// TwinCAT 3 PLC project BaseElements
// Title: Base_Hts
// Company: Vistaprint
// Author: AVME/DSC
// ProjectVersion: 0.0.0.50
// Description: 0.0.0.50 - HFE: Bug fixed 0.0.0.49 - HFE: desable of last station 0.0.0.48 - Add AutoMode to HRU 0.0.0.47 - Some Bugs in DPJ fixed 0.0.0.46 - BaseElements 0.0.1.18 Some Bugs in DPJ, JUN fixed 0.0.0.45 - BaseElements 0.0.1.17 MTR/sta_RUN Bug fixed 0.0.0.44 - New Libs BasePLC 0.3.4.8, BaseElements 0.0.1.16 0.0.0.43 - DPJ reworked (Missed Shirt Problem) 0.0.0.42 - MER - new parameter added HFE reworked 0.0.0.41 - BasePLC V0.3.4.5; BaseElements V0.0.1.9 0.0.0.40 - Add MTR Parameter dinWaitBetweenSensorAndReservation_um 0.0.0.39 - Bug fixed in HFE, CHD; FOC and FOD added 0.0.0.34 - JUN / DPJ replaced with version from Shirtstream 0.0.0.32 - HFE from Lvl1 to Lvl2 and reworked 0.0.0.30 - BaseElements 0.0.1.5 BasePLC 0.3.4.3 included, Tc2_SerialCom 0.0.0.29 - BaseElements 0.0.1.2 BasePLC 0.3.4.2 included; FB_CtrlModule moved to BaseElements 0.0.0.28 - Added ADS data channel to FB_HPS for shirt request from Heatpress 0.0.0.27 - Added bolStopReleaseHangers 0.0.0.26 - DPJ.sta_RUN Entry action reworked 0.0.0.25 - Error JUN changed 0.0.0.24 - Rising Edge detection of bolBringShirt in HPS 0.0.0.23 - HTS, hanger turned line wait at SEP 0.0.0.22 - Bug fixed in STOPbusy 0.0.0.21 - Bugs fixed in HPS 0.0.0.20 - HPS with new Child SEP New BaseElements 0.0.0.20 0.0.0.19 - Alternativ status for run sequence added; Timing reworked in MER jam detection; DPJ STOPBusy reworked, HRU Errors reworked, DPJ new Errors 12 and 13 added 0.0.0.18 - Timeout Run / Stop sequence added 0.0.0.17 - EMO reworked in BaseCtrlModule; CHD "destination full" reworked; AddStpGrp, AddRunGrp removed 0.0.0.16 - Back to BasePLC Lib. V3.3.5 beacuase of PageFaults 0.0.0.15 - Rebuild 0.0.0.14 - Bugzilla ID 03: BufferFull for LineControl added 0.0.0.13 - Bugzilla ID 55: reworked refill of SLB/STB 0.0.0.12 - Update of BasePLC 0.3.3.7, BaseElements 0.0.0.17 0.0.0.11 - Add more controllers to the library (LAI, CHD, HFE, PLS, JUN, DPJ, MER, HRU, HPS, COS, STB, SLB) 0.0.0.10 - Clear pending command to prevent automatic recovery in sta_STOPBusy 0.0.0.9 - BugFix in sub state "cSTA_SUB_CHECK_GROUP_STATUS" from run and stop sequence. Insert new "bolChecked" flag to detect if the sequence has been processed correctly. 0.0.0.8 - Add TSTOP in checkChildAlmClass 0.0.0.7- General revision of behaviour in case of emergency off (state EOFF) and general error (state ERROR). New handling for module specific interface. 0.0.0.6 - Go to EOFFBusy if not in sta_EOFF 0.0.0.5 - In Always: go to EOFFBusy at generalFault 0.0.0.4 - In Always: go to EOFFBusy not to EOFF at emergency stop 0.0.0.3 - Remove CurrentItemCounter and his inputs 0.0.0.2 - Changes after first use in simulation in ICL Module 0.0.0.1 - First release
// ProgramVersion: 3.1.0.5
// libraries:
//   Base_Elements,0.0.1.18,Vistaprint
//   Base_PLC,0.3.4.8,Vistaprint
//   Tc2_Standard,3.3.0.0,Beckhoff Automation GmbH
//   Tc2_System,3.3.5.0,Beckhoff Automation GmbH
//   Tc2_Utilities,3.3.7.0,Beckhoff Automation GmbH
//   Tc3_Module,3.3.5.0,Beckhoff Automation GmbH
// project tree:
//   POUs/Controller/Driver/FOD/ FB_ReceiveFolderState.TcPOU (not stored), FB_SendFolderMessage.TcPOU, T_FOD.TcDUT (not stored), T_FOD_Cfg.TcDUT (not stored), T_FOD_Cur.TcDUT (not stored), T_FOD_StateMachine.TcDUT (not stored)
//   POUs/Controller/Driver/FOD/Infrastructure/ FB_DecodeCanRxMessage.TcPOU (not stored), fb_GenerateCanTxMessage.TcPOU
//   POUs/Controller/Lvl0/CHD %28Cross Hanger Detection%29/ CHD_CmdState.TcGVL (not stored), Const_CHD.TcGVL (not stored), FB_CHD.TcPOU (not stored), T_CheckElement.TcDUT (not stored), T_Ctrl_SIf_CHD.TcDUT (not stored), T_Ctrl_SIf_CHD_Cfg.TcDUT (not stored), T_Ctrl_SIf_CHD_Cur.TcDUT (not stored), T_Ctrl_SIf_CHD_In.TcDUT (not stored), T_Ctrl_SIf_CHD_Out.TcDUT (not stored), T_Ctrl_SIf_CHD_Par.TcDUT (not stored)
//   POUs/Controller/Lvl0/FOC %28Folder Communication%29/ FB_FOC.TcPOU (not stored), FOC_CmdState.TcGVL (not stored), T_Ctrl_SIf_FOC.TcDUT (not stored), T_Ctrl_SIf_FOC_Cfg.TcDUT (not stored), T_Ctrl_SIf_FOC_Cur.TcDUT (not stored), T_Ctrl_SIf_FOC_In.TcDUT (not stored), T_Ctrl_SIf_FOC_Out.TcDUT (not stored), T_Ctrl_SIf_FOC_Par.TcDUT (not stored)
//   POUs/Controller/Lvl0/HRU %28Hanger Rotation Unit%29/ FB_HRU.TcPOU (not stored), HRU_CmdState.TcGVL (not stored), T_Ctrl_SIf_HRU.TcDUT (not stored), T_Ctrl_SIf_HRU_In.TcDUT (not stored), T_Ctrl_SIf_HRU_Out.TcDUT (not stored), T_Ctrl_SIf_HRU_Par.TcDUT (not stored)
//   POUs/Controller/Lvl0/JUN %28Junction%29/ E_Typ_JUN.TcDUT (not stored), FB_JUN.TcPOU (not stored), JUN_CmdState.TcGVL (not stored), T_Ctrl_SIf_JUN.TcDUT (not stored), T_Ctrl_SIf_JUN_Cfg.TcDUT (not stored), T_Ctrl_SIf_JUN_Cur.TcDUT (not stored), T_Ctrl_SIf_JUN_Ilk.TcDUT (not stored), T_Ctrl_SIf_JUN_In.TcDUT (not stored), T_Ctrl_SIf_JUN_Out.TcDUT (not stored), T_Ctrl_SIf_JUN_Par.TcDUT (not stored), T_JUN_OutfeedCheck.TcDUT (not stored)
//   POUs/Controller/Lvl0/LAI %28Labler Interface%29/ FB_LAI.TcPOU (not stored), T_Ctrl_SIf_LAI.TcDUT (not stored), T_Ctrl_SIf_LAI_Cfg.TcDUT (not stored), T_Ctrl_SIf_LAI_Cur.TcDUT (not stored), T_Ctrl_SIf_LAI_In.TcDUT (not stored), T_Ctrl_SIf_LAI_Out.TcDUT (not stored), T_Ctrl_SIf_LAI_Par.TcDUT (not stored)
//   POUs/Controller/Lvl0/PLS %28PickToLight System%29/ Const_PLS.TcGVL (not stored), FB_PLS.TcPOU (not stored), T_Ctrl_SIf_PLS.TcDUT (not stored), T_Ctrl_SIf_PLS_Cfg.TcDUT (not stored), T_Ctrl_SIf_PLS_Cur.TcDUT (not stored), T_Ctrl_SIf_PLS_In.TcDUT (not stored), T_Ctrl_SIf_PLS_Out.TcDUT (not stored), T_Ctrl_SIf_PLS_Par.TcDUT (not stored)
//   POUs/Controller/Lvl0/STB %28Stopper buffer%29/ FB_STB.TcPOU (not stored), STB_CmdState.TcGVL (not stored), T_Ctrl_SIf_STB.TcDUT (not stored), T_Ctrl_SIf_STB_Cfg.TcDUT (not stored), T_Ctrl_SIf_STB_Cur.TcDUT (not stored), T_Ctrl_SIf_STB_Ilk.TcDUT (not stored), T_Ctrl_SIf_STB_In.TcDUT (not stored), T_Ctrl_SIf_STB_Out.TcDUT (not stored), T_Ctrl_SIf_STB_Par.TcDUT (not stored)
//   POUs/Controller/Lvl1/DPJ %28DecisionPoint Junction%29/ Const_DPJ.TcGVL (not stored), DPJ_CmdState.TcGVL (not stored), E_DecisionState.TcDUT (not stored), E_Decision_Job.TcDUT (not stored), E_ProductFlowState.TcDUT (not stored), FB_DPJ.TcPOU (not stored), FB_DtChnToLine_JobDone.TcPOU (not stored), T_Ctrl_SIf_DPJ.TcDUT (not stored), T_Ctrl_SIf_DPJ_Cfg.TcDUT (not stored), T_Ctrl_SIf_DPJ_Cur.TcDUT (not stored), T_Ctrl_SIf_DPJ_DtChnToLine.TcDUT (not stored), T_Ctrl_SIf_DPJ_DtChnToPLC.TcDUT (not stored), T_Ctrl_SIf_DPJ_In.TcDUT (not stored), T_Ctrl_SIf_DPJ_Out.TcDUT (not stored), T_Ctrl_SIf_DPJ_Par.TcDUT (not stored), T_Decision.TcDUT (not stored), T_DecisionElement.TcDUT (not stored), T_Decision_DtChn.TcDUT (not stored), T_JobDone_DtChn.TcDUT (not stored), T_SimDtChn.TcDUT (not stored)
//   POUs/Controller/Lvl1/SLB %28Slide buffer%29/ Const_SLB.TcGVL (not stored), FB_SLB.TcPOU (not stored), SLB_CmdState.TcGVL (not stored), T_Ctrl_SIf_SLB.TcDUT (not stored), T_Ctrl_SIf_SLB_Cfg.TcDUT (not stored), T_Ctrl_SIf_SLB_Cur.TcDUT (not stored), T_Ctrl_SIf_SLB_In.TcDUT (not stored), T_Ctrl_SIf_SLB_Par.TcDUT (not stored)
//   POUs/Controller/Lvl2/COS %28Control Station%29/ COS_CmdState.TcGVL (not stored), FB_COS.TcPOU (not stored), T_Ctrl_SIf_COS.TcDUT (not stored), T_Ctrl_SIf_COS_Cfg.TcDUT (not stored), T_Ctrl_SIf_COS_Cur.TcDUT (not stored), T_Ctrl_SIf_COS_In.TcDUT (not stored), T_Ctrl_SIf_COS_Par.TcDUT (not stored)
//   POUs/Controller/Lvl2/FOL %28Folder%29/ FB_FOL.TcPOU (not stored), FOL_CmdState.TcGVL (not stored), T_Ctrl_SIf_FOL.TcDUT (not stored), T_Ctrl_SIf_FOL_Cfg.TcDUT (not stored), T_Ctrl_SIf_FOL_Cur.TcDUT (not stored), T_Ctrl_SIf_FOL_In.TcDUT (not stored), T_Ctrl_SIf_FOL_Out.TcDUT (not stored), T_Ctrl_SIf_FOL_Par.TcDUT (not stored)
//   POUs/Controller/Lvl2/HFE/ Const_HFE.TcGVL, FB_HFE.TcPOU, T_Ctrl_SIf_HFE.TcDUT, T_Ctrl_SIf_HFE_Cfg.TcDUT, T_Ctrl_SIf_HFE_Cur.TcDUT, T_Ctrl_SIf_HFE_Par.TcDUT
//   POUs/Controller/Lvl2/HPS %28Heat Press Shirt Station%29/ Const_HPS.TcGVL (not stored), E_DtChnJob.TcDUT (not stored), FB_DtChnToLine_ChargeDone.TcPOU (not stored), FB_HPS.TcPOU (not stored), T_ChargeDone_DtChn.TcDUT (not stored), T_Ctrl_SIf_HPS.TcDUT (not stored), T_Ctrl_SIf_HPS_Ads.TcDUT (not stored), T_Ctrl_SIf_HPS_Ads_Read.TcDUT (not stored), T_Ctrl_SIf_HPS_Cfg.TcDUT (not stored), T_Ctrl_SIf_HPS_Cur.TcDUT (not stored), T_Ctrl_SIf_HPS_DtChnToLine.TcDUT (not stored), T_Ctrl_SIf_HPS_DtChnToPLC.TcDUT (not stored), T_Ctrl_SIf_HPS_In.TcDUT (not stored), T_Ctrl_SIf_HPS_Out.TcDUT (not stored), T_Ctrl_SIf_HPS_Par.TcDUT (not stored), T_NewCharge_DtChn.TcDUT (not stored)
//   POUs/Controller/Lvl2/MER %28Merger Standard%29/ Const_MER.TcGVL (not stored), E_Typ_MER_AUTO_MODE.TcDUT (not stored), E_Typ_MER_MODE.TcDUT (not stored), FB_MER.TcPOU (not stored), T_Ctrl_SIf_MER.TcDUT (not stored), T_Ctrl_SIf_MER_Cfg.TcDUT (not stored), T_Ctrl_SIf_MER_Cur.TcDUT (not stored), T_Ctrl_SIf_MER_In.TcDUT (not stored), T_Ctrl_SIf_MER_Par.TcDUT (not stored), T_Line.TcDUT (not stored)
//   POUs/Controller/Lvl2/MTR %28Merger Transport%29/ Const_MTR.TcGVL (not stored), E_Typ_MTR_SECTION_STATE.TcDUT (not stored), FB_MTR.TcPOU (not stored), T_Ctrl_SIf_MTR.TcDUT (not stored), T_Ctrl_SIf_MTR_Cfg.TcDUT (not stored), T_Ctrl_SIf_MTR_Cur.TcDUT (not stored), T_Ctrl_SIf_MTR_In.TcDUT (not stored), T_Ctrl_SIf_MTR_Par.TcDUT (not stored), T_MTR_Buffer_Sections.TcDUT (not stored)
//   Version/ Global_Version.TcGVL
// (motion and I/O tree: see PLC project basehtssample)
// real-time tasks:
//   TASK Task_Fast: cycle T#2ms, priority 3, ADS port 350
//   TASK Task_Slow: cycle T#50000us, priority 20, ADS port 351
//   TASK Task_Middle: cycle T#10ms, priority 10, ADS port 352

// ---- POUs/Controller/Lvl2/HFE/T_Ctrl_SIf_HFE.TcDUT
TYPE T_Ctrl_SIf_HFE :
STRUCT
	///configuration
	Cfg: T_Ctrl_SIf_HFE_Cfg;
	///parameter
	Par: T_Ctrl_SIf_HFE_Par;
	///current values
	Cur: T_Ctrl_SIf_HFE_Cur;
	///alarm number used in this controller
	Alm: ARRAY[1..2] OF T_Ctrl_Alm;
END_STRUCT
END_TYPE

// ---- POUs/Controller/Lvl2/HFE/T_Ctrl_SIf_HFE_Cfg.TcDUT
TYPE T_Ctrl_SIf_HFE_Cfg :
STRUCT
	/// Number of supportetd LDS
	uintNbOfLDS: UINT;
END_STRUCT
END_TYPE

// ---- POUs/Controller/Lvl2/HFE/T_Ctrl_SIf_HFE_Cur.TcDUT
TYPE T_Ctrl_SIf_HFE_Cur :
STRUCT
END_STRUCT
END_TYPE

// ---- POUs/Controller/Lvl2/HFE/T_Ctrl_SIf_HFE_Par.TcDUT
TYPE T_Ctrl_SIf_HFE_Par :
STRUCT
	// Waiting between SLB-STB Close and Junction open
	udiWaitingTime_ms: UDINT;
	// Open junction time
	a_udiTimeOpen_ms: ARRAY[0..cuintMaxStation] OF UDINT;
	// Close junction time
	a_udiTimeClose_ms: ARRAY[0..cuintMaxStation] OF UDINT;
	// Enable Junction to LDS
	a_bolEnableJunction: ARRAY[0..cuintMaxStation] OF BOOL;
END_STRUCT
END_TYPE

// ---- POUs/Controller/Lvl2/HFE/Const_HFE.TcGVL
VAR_GLOBAL CONSTANT
	cuintMaxStation: INT := 4;
END_VAR

// ---- Version/Global_Version.TcGVL
// This function has been automatically generated from the project information.
VAR_GLOBAL CONSTANT
	{attribute 'const_non_replaced'}
	stLibVersion_Base_Hts : ST_LibVersion := (iMajor := 0, iMinor := 0, iBuild := 0, iRevision := 50, sVersion := '0.0.0.50');
END_VAR

// ---- POUs/Controller/Driver/FOD/FB_SendFolderMessage.TcPOU
FUNCTION_BLOCK FB_SendFolderMessage
VAR_INPUT
	InTxCounter AT %I*: UINT;
	CpuOnline: BOOL;
	EmptyHangerConveying: BOOL;
	ProgramNumber: BYTE := 1;
	/// 1=forward, 2=sideward
	ShirtStackConveyor: BYTE := 1;
	ChangeCustomer: BOOL;
	StopFolder: BOOL;
	ShotOutStacks: BOOL;
	/// CAN Identifier of receiver
	TxCobId: UINT := 113;
	/// true = starts sending a message. make sure all data fields are set before.
	bStartSend: BOOL;
	/// timeout after sent message before next message will be send
	tTimeout: TIME := TIME#50ms;
END_VAR
VAR_OUTPUT
	TxMessages AT %Q*: ARRAY[0..9] OF CANQUEUE;
	OutTxCounter AT %Q*: UINT;
	OutNoOfTxMessages AT %Q*: UINT := 1;
END_VAR
VAR
	uinState: UINT;
	BytesToSend: UINT := 8;
	arrDataToSend: CANMESSAGE;
	m: UINT;
	fbGenerateTxMessage: fb_GenerateCanTxMessage;
	uliCountSentMessages: ULINT;
	tWaitTimer: TON;
END_VAR
VAR CONSTANT
	cSTA_WAIT_SEND: UINT := 10;
	cSTA_SEND_MESSAGE: UINT := 20;
	cSTA_WAIT_SEND_COMPLETE: UINT := 30;
	cSTA_WAIT_BEFORE_SEND_NEXT: UINT := 40;
END_VAR

(*__________________________________________________________________________________________________
¦	
¦	Vistaprint Schweiz GmbH
¦	CH - 8401 Winterthur
¦
¦	www.vistaprint.ch - info@vistaprint.ch
¦___________________________________________________________________________________________________

Function desription:
CAN communication to Kannegiesser folder to send commands.


History:
Version		Date			Author		Comment
---------------------------------------------------------------------------------------------------
0.00.1		28.09.2013		VP/RE		Start history
0.00.2		29.10.2013		VP/RE		Introduced state names
0.00.3		11.12.2013		VP/RE		Implemented sleep timeout after sending a CAN message.
___________________________________________________________________________________________________*)


CASE uinState OF
	
cSTA_WAIT_SEND:	
	IF bStartSend THEN
		bStartSend:=FALSE;
		uinState := cSTA_SEND_MESSAGE;
	END_IF
	
cSTA_SEND_MESSAGE:	
	
	uliCountSentMessages := uliCountSentMessages + 1;

	FOR m := 0 TO OutNoOfTxMessages - 1 DO
		
		arrDataToSend[0].0 := CpuOnline;
		arrDataToSend[0].1 := EmptyHangerConveying;
		arrDataToSend[1].0 := ChangeCustomer;
		
		arrDataToSend[0].4 := ProgramNumber.0;
		arrDataToSend[0].5 := ProgramNumber.1;
		arrDataToSend[0].6 := ProgramNumber.2;
		arrDataToSend[0].7 := ProgramNumber.3;
		
		IF (ShirtStackConveyor = 1) THEN
			arrDataToSend[2].1 := 1;
			arrDataToSend[2].2 := 0;
		ELSIF (ShirtStackConveyor = 2) THEN
			arrDataToSend[2].1 := 0;
			arrDataToSend[2].2 := 1;
		ELSIF (ShirtStackConveyor = 0) THEN
			arrDataToSend[2].1 := 0;
			arrDataToSend[2].2 := 0;
		END_IF
		
		arrDataToSend[3].5 := StopFolder;
		arrDataToSend[3].6 := ShotOutStacks;

		fbGenerateTxMessage(CobId := TxCobId,
							BytesToSend := BytesToSend,
							arrDataToSend := arrDataToSend ,
							TxMessage => TxMessages[0] );
	END_FOR
	
	OutTxCounter := OutTxCounter + 1;
	uinState := cSTA_WAIT_SEND_COMPLETE;
	
cSTA_WAIT_SEND_COMPLETE:	
	IF OutTxCounter = InTxCounter THEN
		uinState := cSTA_WAIT_BEFORE_SEND_NEXT;
	END_IF

cSTA_WAIT_BEFORE_SEND_NEXT:
	IF (tWaitTimer.Q = TRUE) THEN
		uinState := cSTA_WAIT_SEND;
	END_IF
	
END_CASE

tWaitTimer(IN := uinState = cSTA_WAIT_BEFORE_SEND_NEXT, PT := tTimeout);

METHOD init
uinState := cSTA_WAIT_SEND;
END_METHOD

END_FUNCTION_BLOCK

// ---- POUs/Controller/Driver/FOD/Infrastructure/fb_GenerateCanTxMessage.TcPOU
FUNCTION_BLOCK fb_GenerateCanTxMessage
VAR_INPUT
	CobId: UINT;
	BytesToSend: UINT;
	arrDataToSend: CANMESSAGE;
END_VAR
VAR_OUTPUT
	TxMessage: CANQUEUE;
END_VAR

TxMessage.CobId := (SHL(CobId,5)) + BytesToSend;
TxMessage.data := arrDataToSend;

END_FUNCTION_BLOCK

// ---- POUs/Controller/Lvl2/HFE/FB_HFE.TcPOU
FUNCTION_BLOCK FB_HFE EXTENDS FB_CtrlBase
VAR_INPUT
	a_bolLDSNeedsHanger: ARRAY[0..cuintMaxStation] OF BOOL;
	a_intHFE_BufferZone: ARRAY[0..cuintMaxStation] OF INT;
	p_fbTlpDrive: POINTER TO FB_DRV;
	///p_fbJunction : POINTER TO FB_JUN;
	p_fbSLB: POINTER TO FB_SLB;
END_VAR
VAR
	/// List of pointers to Childs of VLV
	a_pMultiChildCtrl: ARRAY[0..Base_Const.cMaxNrOfChilds] OF POINTER TO FB_VLV;
	/// List of childs common interface
	a_pMultiChildCIF: ARRAY[0..Base_Const.cMaxNrOfChilds] OF POINTER TO T_Ctrl_CIf;
	/// List of childs specific interface for additional parameters or cur
	a_pMultiChildSIF: ARRAY[0..Base_Const.cMaxNrOfChilds] OF POINTER TO Base_Elements.T_Ctrl_SIf_VLV;
	usiNumOfMultiChild: USINT;
	usiNumOfValidPointerMultiChild: USINT;
	/// Specific interface struct for public access
	SIf: T_Ctrl_SIf_HFE;
	/// Child controller
	pTlpDrive_CIf: POINTER TO T_Ctrl_CIf;
	///pJunction_CIf : POINTER TO T_Ctrl_CIf;
	pSLB_CIf: POINTER TO T_Ctrl_CIf;
	pSLB_SIf: POINTER TO T_Ctrl_SIf_SLB;
	intSubState: ARRAY[0..cuintMaxStation] OF INT;
	udiTimeInStateRefill_ms: ARRAY[0..cuintMaxStation] OF UDINT;
END_VAR
VAR CONSTANT
	/// sub States
	cSTA_SUB_WaitForJob: INT := 500;
	cSTA_SUB_WaitOpen: INT := 502;
	cSTA_SUB_Open: INT := 504;
	cSTA_SUB_WaitClose: INT := 506;
	cSTA_SUB_Close: INT := 508;
END_VAR

(*__________________________________________________________________________________________________
¦	
¦	Vistaprint Schweiz GmbH
¦	CH - 8401 Winterthur
¦
¦	www.vistaprint.ch - info@vistaprint.ch
¦___________________________________________________________________________________________________

Function desription:
Cylinder implementation. 


History:
Version		Date			Author		Comment
---------------------------------------------------------------------------------------------------
0.00.1		02.07.2013		VP/RE		Start history
0.00.2		16.12.2013		AVME/MRU	In Always: No EOFF State!! in EOFF go to OFF

___________________________________________________________________________________________________*)



// check if child pointer valid
IF (me.bolActivate) AND (p_fbTlpDrive<>0)  AND (THIS^.checkChildPointer()) AND (p_fbSLB<>0) THEN // cyclic call enabled
	
	IF (CIf.Info.bolInitDone=FALSE) THEN // first cycle -> init
		CtrlInit();
		CIf.Info.bolInitDone := TRUE;
	ELSE
		CycleStartDuty();
	
		Always();
		
		StateMachine();
		
		CycleEndDuty();
	END_IF
	
END_IF;

METHOD PROTECTED checkChildPointer : BOOL
IF (usiNumOfMultiChild = usiNumOfValidPointerMultiChild) THEN
	checkChildPointer:= TRUE;
ELSE
	checkChildPointer:= FALSE;
END_IF
END_METHOD

METHOD PROTECTED StateMachine : BOOL
SUPER^.StateMachine();

// main statemachine of base controller
CASE me.StateMachine.intState OF
	 cSTA_RUN: 
        THIS^.sta_RUN();
	cSTA_RUNBusy:
        THIS^.sta_RUNBusy();
END_CASE;
END_METHOD

METHOD PROTECTED Always : BOOL
SUPER^.Always();

IF (me.StateMachine.intState<>cSTA_SINGLE_ANSWER) THEN
	
	;
	
END_IF

// ----------------------------------------------------------------------------------
// Conditions Always
// overrule error always from base -> no EOFF State!! in EOFF go to OFF
IF (me.StateMachine.intStateNext = cSTA_EOFFBusy) THEN
	IF (me.StateMachine.intState=cSTA_OFF) THEN
		me.StateMachine.intStateNext := cSTA_OFF;
	ELSE // stay in OFF
		me.StateMachine.intStateNext := cSTA_OFFBusy;
	END_IF
END_IF
END_METHOD

METHOD AddJunction
VAR_INPUT
	p_MultiChild: POINTER TO FB_JUN;
END_VAR

// Method add the pointer address of the buffer zone child controller to the array list.
IF (usiNumOfMultiChild <= (Base_Const.cMaxNrOfChilds-1)) THEN
	// Add buffer zone child controller to list
	a_pMultiChildCtrl[usiNumOfMultiChild] := p_MultiChild;
	// Inc. number of buffer zones
	usiNumOfMultiChild:= usiNumOfMultiChild+1;
	// Check if the pointer is valid
	IF (p_MultiChild<>0) THEN
		usiNumOfValidPointerMultiChild:= usiNumOfValidPointerMultiChild+1;
	END_IF
END_IF
END_METHOD

METHOD getCtrlSIf : POINTER TO T_Ctrl_SIf_HFE
getCtrlSIf := ADR(SIf);
END_METHOD

METHOD PROTECTED sta_OFF : BOOL
// state implemetation
//--------------------------------------------------------------------------------------
// Entry action
	IF (me.StateMachine.intState<>me.StateMachine.intStateLastCycle) THEN
		me.StateMachine.intStateLastCycle := me.StateMachine.intState;
		
	END_IF


//--------------------------------------------------------------------------------------
// Cyclic action
	IF (me.StateMachine.intState=me.StateMachine.intStateLastCycle) THEN
		
		;
		
		// State Change Condition
		IF me.intCmd=cCMD_RUN THEN
			me.StateMachine.intStateNext :=  cSTA_RUNBusy;
		END_IF
	END_IF




//--------------------------------------------------------------------------------------
// Exit action
	IF (me.StateMachine.intState<>me.StateMachine.intStateNext) THEN
		;
	END_IF
END_METHOD

METHOD PROTECTED IoOutBridge : BOOL
VAR
	bolSwitchValvesOff: BOOL;
END_VAR
// digitale and analoge inputs read from hardware or forcing
IF (CIf.SwCfg.bolSimulation = FALSE) THEN
	//setOutBol(CIf.Job.bolIoForce ,ADR(SIf.Out.bolClamping));

	//THIS^.Out_Clamping := SIf.Out.bolClamping.map;
END_IF
END_METHOD

METHOD PROTECTED IoInBridge : BOOL
// digitale and analoge inputs read from hardware or forcing
//SIf.In.bolGiveNextHangerSensor.map := THIS^.In_GiveNextHangerSensor;

IF (CIf.SwCfg.bolSimulation = FALSE) THEN
	//getInBol(CIf.Job.bolIoForce,ADR(SIf.In.bolGiveNextHangerSensor));
ELSE
	//simulation of global IO
END_IF
END_METHOD

METHOD PROTECTED sta_RUNBusy : BOOL
// state implemetation
//--------------------------------------------------------------------------------------
// Entry action
	IF (me.StateMachine.intState<>me.StateMachine.intStateLastCycle) THEN
		me.StateMachine.intStateLastCycle := me.StateMachine.intState;
		
		pTlpDrive_CIf^.Job.intACmd := cCMD_RUN;
		pSLB_CIf^.Job.intACmd := Base_PLC.cCMD_RUN;
		
	END_IF


//--------------------------------------------------------------------------------------
// Cyclic action
	IF (me.StateMachine.intState=me.StateMachine.intStateLastCycle) THEN
		
		// State Change Condition
		IF (pTlpDrive_CIf^.Job.intState = cSTA_RUN) THEN
			me.StateMachine.intStateNext := cSTA_RUN;
		END_IF
	END_IF



//--------------------------------------------------------------------------------------
// Exit action
	IF (me.StateMachine.intState<>me.StateMachine.intStateNext) THEN
		;
	END_IF
END_METHOD

METHOD Refill
VAR_INPUT
	intNbOfLDS: INT;
END_VAR
VAR
	/// Loop variable
	ii: INT;
END_VAR
// Simulation
fbSimulationTimer.PT := UDINT_TO_TIME(1000);
IF (CIf.SwCfg.bolSimulation) THEN
	// Cyclicle input into the top stopperbuffer
	fbSimulationTimer(); // set time/reset timer
	IF fbSimulationTimer.Q = TRUE THEN
		fbSimulationTimer.IN := FALSE;
	ELSE
		fbSimulationTimer.IN := TRUE;
	END_IF
			
END_IF

// Method refill 
CASE intSubState[intNbOfLDS] OF
	cSTA_SUB_WaitForJob: // LDS needs hanger
		IF (a_bolLDSNeedsHanger[intNbOfLDS]) THEN
//			IF (p_fbSLB^.CtrlCIf^.Info.p_aCIf[intNbOfLDS + 2]^.job.intState = 6) OR (p_fbSLB^.CtrlCIf^.Info.p_aCIf[intNbOfLDS + 2]^.job.intState = 12) THEN //	Just open if PreStopper is closed
			IF (p_fbSLB^.CtrlCIf^.Info.p_aCIf[a_intHFE_BufferZone[intNbOfLDS]]^.job.intState = 6) 
			OR (p_fbSLB^.CtrlCIf^.Info.p_aCIf[a_intHFE_BufferZone[intNbOfLDS]]^.job.intState = 12) THEN //	Just open if PreStopper is closed
				a_pMultiChildCIF[intNbOfLDS]^.Job.intACmd:= Base_Elements.VLV_CmdState.cCMD_OPEN;
				udiTimeInStateRefill_ms[intNbOfLDS] := 0;
				intSubState[intNbOfLDS] := cSTA_SUB_WaitOpen;
			END_IF
		END_IF
	
	cSTA_SUB_WaitOpen:	// Waiting time between STB closing and junction opening
		udiTimeInStateRefill_ms[intNbOfLDS]:= udiTimeInStateRefill_ms[intNbOfLDS] + me.FUBInfo.udiSample_ms;
		IF (udiTimeInStateRefill_ms[intNbOfLDS] > SIf.Par.udiWaitingTime_ms) THEN
			intSubState[intNbOfLDS] := cSTA_SUB_Open;
			udiTimeInStateRefill_ms[intNbOfLDS] := 0;			
		END_IF
		
	cSTA_SUB_Open:	
		udiTimeInStateRefill_ms[intNbOfLDS]:= udiTimeInStateRefill_ms[intNbOfLDS] + me.FUBInfo.udiSample_ms;
		IF ((Sif.Par.a_udiTimeOpen_ms[intNbOfLDS] <> 0) AND (Sif.Par.a_udiTimeOpen_ms[intNbOfLDS] < udiTimeInStateRefill_ms[intNbOfLDS])) OR 
		(a_bolLDSNeedsHanger[intNbOfLDS] = 0) THEN
			intSubState[intNbOfLDS] := cSTA_SUB_WaitClose;
		END_IF
		
	cSTA_SUB_WaitClose:	// Waiting time between STB closing and junction closing
//		IF (p_fbSLB^.CtrlCIf^.Info.p_aCIf[intNbOfLDS + 2]^.job.intState = 6) or (p_fbSLB^.CtrlCIf^.Info.p_aCIf[intNbOfLDS + 2]^.job.intState = 12) THEN //	Just close if PreStopper is closed
		IF (p_fbSLB^.CtrlCIf^.Info.p_aCIf[a_intHFE_BufferZone[intNbOfLDS]]^.job.intState = 6) 
		OR (p_fbSLB^.CtrlCIf^.Info.p_aCIf[a_intHFE_BufferZone[intNbOfLDS]]^.job.intState = 12) THEN //	Just close if PreStopper is closed

			udiTimeInStateRefill_ms[intNbOfLDS] := 0;
			intSubState[intNbOfLDS] := cSTA_SUB_Close;
		END_IF
		
	cSTA_SUB_Close:
		udiTimeInStateRefill_ms[intNbOfLDS]:= udiTimeInStateRefill_ms[intNbOfLDS] + me.FUBInfo.udiSample_ms;
		IF (udiTimeInStateRefill_ms[intNbOfLDS] > SIf.Par.udiWaitingTime_ms) THEN
			a_pMultiChildCIF[intNbOfLDS]^.Job.intACmd:= Base_Elements.VLV_CmdState.cCMD_Close;
			IF ((Sif.Par.a_udiTimeClose_ms[intNbOfLDS] < udiTimeInStateRefill_ms[intNbOfLDS])) THEN
				intSubState[intNbOfLDS] := cSTA_SUB_WaitForJob;
			END_IF
		END_IF
END_CASE
END_METHOD

METHOD PROTECTED sta_RUN : BOOL
VAR
	intNbOfLDS: INT;
	intI: INT;
END_VAR
// state implemetation
//--------------------------------------------------------------------------------------
// Entry action
	IF (me.StateMachine.intState<>me.StateMachine.intStateLastCycle) THEN
		me.StateMachine.intStateLastCycle := me.StateMachine.intState;
		
		//fbSimulationTimer.IN := FALSE;
		//fbSimulationTimer.PT := UDINT_TO_TIME(SIf.Par.udi_pulseTimeout_ms/10);
		//fbSimulationTimer(); // set time/reset timer
		//fbSimulationTimer.IN := TRUE; // start timer
		FOR intNbOfLDS := 0 TO UINT_TO_INT(cuintMaxStation) DO
			intSubState[intNbOfLDS] := 500;	// Init Refill Substate
		END_FOR
	END_IF


//--------------------------------------------------------------------------------------
// Cyclic action
	IF (me.StateMachine.intState=me.StateMachine.intStateLastCycle) THEN
		
		// Simulation
		IF (CIf.SwCfg.bolSimulation) THEN
			//fbSimulationTimer(); // simulation time
			//IF (fbSimulationTimer.Q) THEN
			//	SIf.In.bolPulse.intern := NOT SIf.In.bolPulse.intern; // toggle pulse
			//	fbSimulationTimer.IN := FALSE;
			//ELSE
			//	fbSimulationTimer.IN := TRUE;
			//END_IF
		END_IF
		
		//IF NOT(pSLB_SIf^.Cur.bolBufferFull) THEN
		//	pStopperBuffer_CIf^.Job.intACmd := STB_CmdState.cCMD_RELEASE;
		//END_IF
		FOR intNbOfLDS := 0 TO UINT_TO_INT(cuintMaxStation) DO
			IF (SIf.Par.a_bolEnableJunction[intNbOfLDS]) AND (a_pMultiChildCtrl[intNbOfLDS]<>0) THEN
				Refill(intNbOfLDS);
			END_IF
			IF (INT_TO_UINT(intNbOfLDS) = (SIf.Cfg.uintNbOfLDS-1)) THEN // Last station = End of SLB, no VLV there

				IF (SIf.Par.a_bolEnableJunction[intNbOfLDS] = FALSE) THEN 			// Last Station is unused
					FOR intI := 0 TO UINT_TO_INT(SIf.Cfg.uintNbOfLDS-1) DO
						IF (SIf.Par.a_bolEnableJunction[intNbOfLDS-intI] = TRUE) THEN	// Find last used Station
							a_pMultiChildCIF[intNbOfLDS-intI]^.Job.intACmd:= Base_Elements.VLV_CmdState.cCMD_OPEN;	// Close last Junction
							EXIT;	// Last used Junction found, exit loop
						ELSE															
							IF (INT_TO_UINT(intI) = (SIf.Cfg.uintNbOfLDS-1)) THEN					// No Station is enabled
								// Set Alarm: SIf.Alm[1].strText := 'No Station is enabled!'; 
								pfbAlarmCtrl^.setAlarm(CIf.Info.intCtrlId,1,0,ADR(SIf.Alm),E_AlmState.RST,CIf.Job.eMe_ActivAlmClass);
							END_IF
						END_IF
					END_FOR
				ELSE	// Last Station is enabled -> Normal Work 
					IF (a_bolLDSNeedsHanger[intNbOfLDS]= TRUE) THEN
						IF (pSLB_SIf^.Cur.bolHangerDetected = TRUE) THEN // Just if Hanger is at Last STB
							pSLB_CIf^.Job.intACmd := SLB_CmdState.cCMD_RELEASE;	
						END_IF
					END_IF					
				END_IF
			END_IF
		END_FOR
		
		// State Change Condition
		IF me.intCmd=cCMD_OFF THEN
			me.StateMachine.intStateNext := cSTA_OFFBusy;
		END_IF
		
	END_IF



//--------------------------------------------------------------------------------------
// Exit action
	IF (me.StateMachine.intState<>me.StateMachine.intStateNext) THEN
		;
	END_IF
END_METHOD

METHOD PROTECTED CtrlInit : BOOL
VAR
	ii: INT;
END_VAR
SUPER^.CtrlInit();

// get child CIf
pTlpDrive_CIf := THIS^.AddChild(p_fbTlpDrive^);
pSLB_CIf := THIS^.AddChild(p_fbSLB^);
pSLB_SIf := p_fbSLB^.getCtrlSIf();

//initialize all multi Child controller.
FOR ii:=0 TO usiNumOfMultiChild-1 BY 1 DO	
	// Get child common if
	a_pMultiChildCIF[ii]:= THIS^.AddChild(a_pMultiChildCtrl[ii]^);	
	// Get specific interface for additional parmaeters or cur
	a_pMultiChildSIF[ii]:= a_pMultiChildCtrl[ii]^.getCtrlSIf();
END_FOR
END_METHOD

METHOD FB_init : BOOL
VAR_INPUT
	///if TRUE, the retain variables are initialized (warm start / cold start)
	bInitRetains: BOOL;
	///if TRUE, the instance afterwards gets moved into the copy code (online change)
	bInCopyCode: BOOL;
END_VAR
VAR
	ii: UINT;
END_VAR
//------------------------------------------------------------------------------------------------------------------------
// to manually change in new FUB implementation!!!
// define valid commands for this controller
FOR ii:= 0 TO (SIZEOF(CIf.Job.aCmdList)/SIZEOF(CIf.Job.aCmdList[0])-1) BY 1 DO
	IF (CIf.Job.aCmdList[ii].intCmd=cCMD_INITIALIZED) THEN
		// found first empty array element
		EXIT;
	END_IF
END_FOR
CIf.Job.aCmdList[ii].intCmd := cCMD_RUN;
CIf.Job.aCmdList[ii].strName := 'Run'; 
CIf.Job.aCmdList[ii].bolAvailable := TRUE;
//ii := ii +1;
//CIf.Job.aCmdList[ii].intCmd := cCMD_RETRACT;
//CIf.Job.aCmdList[ii].strName := 'Retract';
//CIf.Job.aCmdList[ii].bolAvailable := TRUE;

// set name of class/typ
CIf.Info.strType := 'FB_HFE'; 

// set alarm class
SIf.Alm[1].eAlmClass := E_AlmClass.INFO;
SIf.Alm[1].strText := 'No Station is enabled!'; 
//SIf.Alm[2].eAlmClass := E_AlmClass.STOP;
//SIf.Alm[2].strText := 'Emergency button pressed.'; 

//*******************************************************************************
// initial values
//*******************************************************************************

// software configuration
CIf.SwCfg.bolExist := TRUE;
CIf.SwCfg.bolSimulation := FALSE;

// parmeter
FOR ii:= 0 TO cuintMaxStation DO
	SIf.Par.a_udiTimeClose_ms[ii] := 10000;
	SIf.Par.a_udiTimeOpen_ms[ii] := 10000;
END_FOR
SIf.Par.udiWaitingTime_ms := 100;
SIf.Par.a_bolEnableJunction[0] := TRUE; // First LDS is enabled

// configuration
SIf.Cfg.uintNbOfLDS := 1;

// actual values
//SIf.Cur.dinCounter := 0;
END_METHOD

END_FUNCTION_BLOCK
